// TwinCAT 3 PLC project PlcFormat
// ProgramVersion: 3.1.4024.0
// libraries:
//   Tc2_Utilities, * (Beckhoff Automation GmbH)
// project tree:
//   POUs/ MAIN.TcPOU

// ---- POUs/MAIN.TcPOU
PROGRAM MAIN
VAR
    measured : LREAL;
    display : STRING;
END_VAR

measured := measured + 0.125;
display := LREAL_TO_FMTSTR(measured, 2, TRUE);

END_PROGRAM
